// TIA Portal project "2022.04.27_指示灯依次亮灭" (V17)

(* hardware
DEVICE "S7-1500/ET200MP station_1"  S7-1500 station
   slot 0: "导轨_0"  Rack  6ES7 590-1***0-0AA0
   slot 1: "PLC_1"  CPU 1516-3 PN/DP  6ES7 516-3AN00-0AB0  V1.7
      slot 3: "CPU 显示_1"  6ES7591-1BA00-0AA0
      slot 32768: "PROFINET 接口_1"  X1
         slot 32769: "端口_1"  X1 P1
         slot 32770: "端口_2"  X1 P2
      slot 33024: "PROFINET 接口_2"  X2
         slot 33025: "端口_1"  X2 P1
      slot 33280: "DP 接口_1"  X3
   slot 2: "DI 32x24VDC BA_1"  DI 32x24VDC BA  6ES7 521-1BL10-0AA0  V1.1
   slot 3: "DQ 32x24VDC/0.5A HF_1"  DQ 32x24VDC/0.5A HF  6ES7 522-1BL01-0AB0  V1.1
*)

// ===== PLC "PLC_1"  CPU 1516-3 PN/DP =====

VAR_GLOBAL   // PLC tag table "默认变量表"
   "亮灯按钮" AT %I0.0 : Bool;
   "灭灯按钮" AT %I0.1 : Bool;
   "复位" AT %I0.2 : Bool;
   "按钮4" AT %I0.3 : Bool;
   "按钮5" AT %I0.4 : Bool;
   "按钮6" AT %I0.5 : Bool;
   "按钮7" AT %I0.6 : Bool;
   "按钮8" AT %I0.7 : Bool;
   "按钮9" AT %I1.0 : Bool;
   "按钮10" AT %I1.1 : Bool;
   "按钮11" AT %I1.2 : Bool;
   "指示灯1" AT %Q0.0 : Bool;
   "指示灯2" AT %Q0.1 : Bool;
   "指示灯3" AT %Q0.2 : Bool;
   "指示灯4" AT %Q0.3 : Bool;
   "指示灯5" AT %Q0.4 : Bool;
   "指示灯6" AT %Q0.5 : Bool;
   "指示灯7" AT %Q0.6 : Bool;
   "指示灯8" AT %Q0.7 : Bool;
   "指示灯9" AT %Q1.0 : Bool;
   "指示灯10" AT %Q1.1 : Bool;
   "指示灯11" AT %Q1.2 : Bool;
   "指示灯12" AT %Q1.3 : Bool;
END_VAR

DATA_BLOCK "计数亮灯LAD_DB"   // DB1
{ S7_Optimized_Access := 'TRUE' }
VERSION : 0.1
// stored: InstanceOfName 计数亮灯LAD
"计数亮灯LAD"
BEGIN
END_DATA_BLOCK

DATA_BLOCK "计数亮灯LAD_DB_1"   // DB3
{ S7_Optimized_Access := 'TRUE' }
VERSION : 0.1
// stored: InstanceOfName 计数亮灯LAD
"计数亮灯LAD"
BEGIN
END_DATA_BLOCK

DATA_BLOCK "计数亮灯FBD_DB"   // DB4
{ S7_Optimized_Access := 'TRUE' }
VERSION : 0.1
// stored: InstanceOfName 计数亮灯FBD
"计数亮灯FBD"
BEGIN
END_DATA_BLOCK

DATA_BLOCK "计数器SCL_DB"   // DB5
{ S7_Optimized_Access := 'TRUE' }
VERSION : 0.1
// stored: InstanceOfName 计数器SCL
"计数器SCL"
BEGIN
END_DATA_BLOCK

// folder: System blocks/Program resources

DATA_BLOCK "IEC_Counter_0_DB"   // DB2
{ S7_Optimized_Access := 'TRUE' }
AUTHOR : Simatic
FAMILY : IEC
NAME : CNTR
VERSION : 1.0
// stored: InstanceOfName IEC_COUNTER
"IEC_COUNTER"
BEGIN
END_DATA_BLOCK

// folder: (top level)

FUNCTION_BLOCK "计数亮灯LAD"   // FB1, LAD
{ S7_Optimized_Access := 'TRUE' }
VERSION : 0.1
   VAR RETAIN
      IEC_Counter_0_Instance : CTUD_INT;
      IEC_Counter_0_Instance_1 : CTUD_INT;
      IEC_Counter_0_Instance_2 : CTUD_INT;
      IEC_Counter_0_Instance_3 : CTUD_INT;
      IEC_Counter_0_Instance_4 : CTUD_INT;
      IEC_Counter_0_Instance_5 : CTUD_INT;
      IEC_Counter_0_Instance_6 : CTUD_INT;
      IEC_Counter_0_Instance_7 : CTUD_INT;
      IEC_Counter_0_Instance_8 : CTUD_INT;
      IEC_Counter_0_Instance_9 : CTUD_INT;
      IEC_Counter_0_Instance_10 : CTUD_INT;
      IEC_Counter_0_Instance_11 : CTD_INT;
   END_VAR
BEGIN

REGION Network 1: 亮灯按钮:选择置位，前灯亮和后灯不亮. 灭灯按钮：复位后灯依次不亮
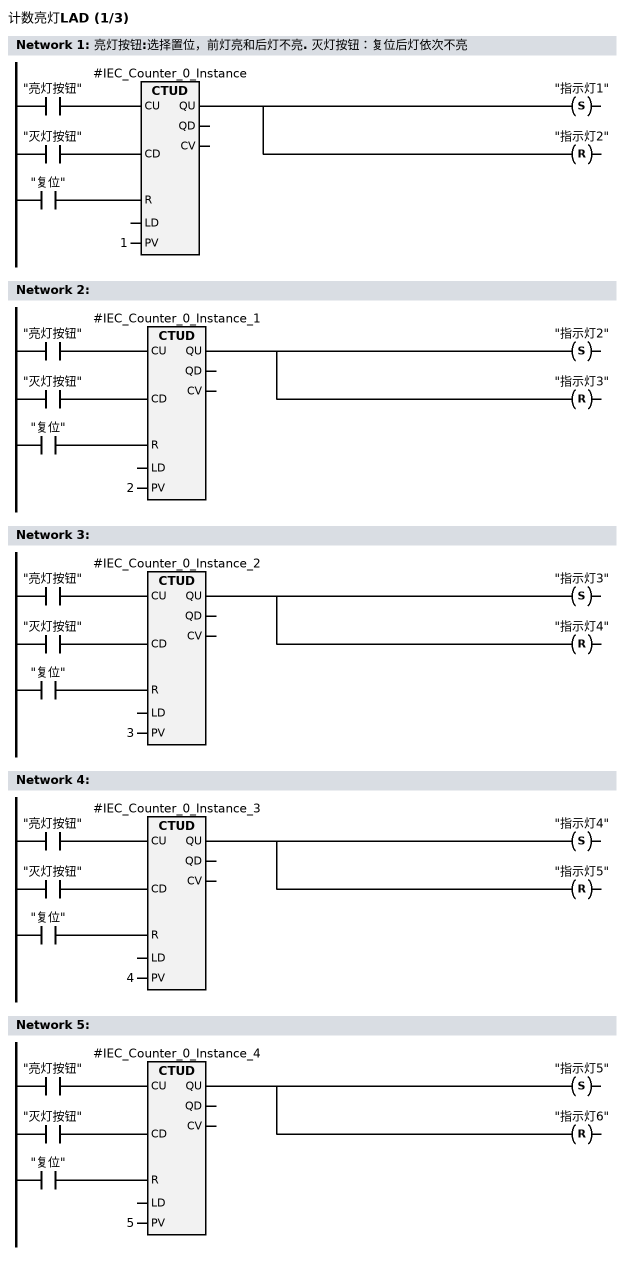
   #IEC_Counter_0_Instance(CU := "亮灯按钮", CD := "灭灯按钮", R := "复位", PV := 1);   // CTUD
   IF #IEC_Counter_0_Instance.QU THEN
       "指示灯1" := TRUE;
       "指示灯2" := FALSE;
   END_IF;
END_REGION

REGION Network 2
   #IEC_Counter_0_Instance_1(CU := "亮灯按钮", CD := "灭灯按钮", R := "复位", PV := 2);   // CTUD
   IF #IEC_Counter_0_Instance_1.QU THEN
       "指示灯2" := TRUE;
       "指示灯3" := FALSE;
   END_IF;
END_REGION

REGION Network 3
   #IEC_Counter_0_Instance_2(CU := "亮灯按钮", CD := "灭灯按钮", R := "复位", PV := 3);   // CTUD
   IF #IEC_Counter_0_Instance_2.QU THEN
       "指示灯3" := TRUE;
       "指示灯4" := FALSE;
   END_IF;
END_REGION

REGION Network 4
   #IEC_Counter_0_Instance_3(CU := "亮灯按钮", CD := "灭灯按钮", R := "复位", PV := 4);   // CTUD
   IF #IEC_Counter_0_Instance_3.QU THEN
       "指示灯4" := TRUE;
       "指示灯5" := FALSE;
   END_IF;
END_REGION

REGION Network 5
   #IEC_Counter_0_Instance_4(CU := "亮灯按钮", CD := "灭灯按钮", R := "复位", PV := 5);   // CTUD
   IF #IEC_Counter_0_Instance_4.QU THEN
       "指示灯5" := TRUE;
       "指示灯6" := FALSE;
   END_IF;
END_REGION

REGION Network 6
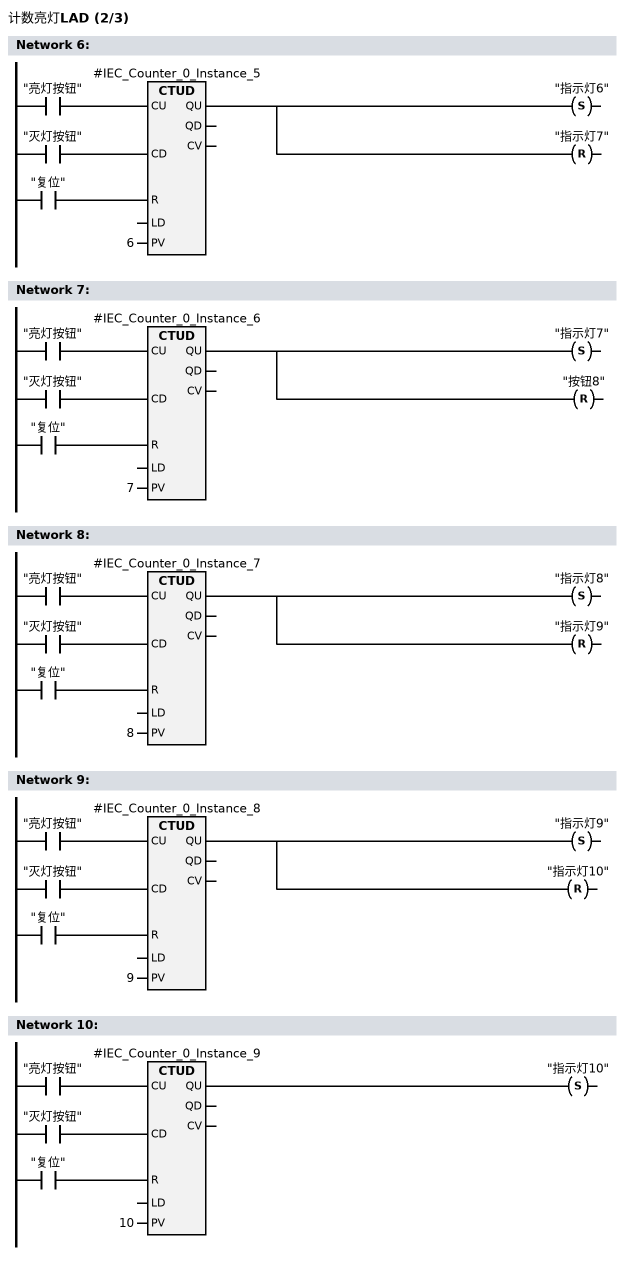
   #IEC_Counter_0_Instance_5(CU := "亮灯按钮", CD := "灭灯按钮", R := "复位", PV := 6);   // CTUD
   IF #IEC_Counter_0_Instance_5.QU THEN
       "指示灯6" := TRUE;
       "指示灯7" := FALSE;
   END_IF;
END_REGION

REGION Network 7
   #IEC_Counter_0_Instance_6(CU := "亮灯按钮", CD := "灭灯按钮", R := "复位", PV := 7);   // CTUD
   IF #IEC_Counter_0_Instance_6.QU THEN
       "指示灯7" := TRUE;
       "按钮8" := FALSE;
   END_IF;
END_REGION

REGION Network 8
   #IEC_Counter_0_Instance_7(CU := "亮灯按钮", CD := "灭灯按钮", R := "复位", PV := 8);   // CTUD
   IF #IEC_Counter_0_Instance_7.QU THEN
       "指示灯8" := TRUE;
       "指示灯9" := FALSE;
   END_IF;
END_REGION

REGION Network 9
   #IEC_Counter_0_Instance_8(CU := "亮灯按钮", CD := "灭灯按钮", R := "复位", PV := 9);   // CTUD
   IF #IEC_Counter_0_Instance_8.QU THEN
       "指示灯9" := TRUE;
       "指示灯10" := FALSE;
   END_IF;
END_REGION

REGION Network 10
   #IEC_Counter_0_Instance_9(CU := "亮灯按钮", CD := "灭灯按钮", R := "复位", PV := 10);   // CTUD
   IF #IEC_Counter_0_Instance_9.QU THEN "指示灯10" := TRUE; END_IF;
END_REGION

REGION Network 11: 复位指示灯1
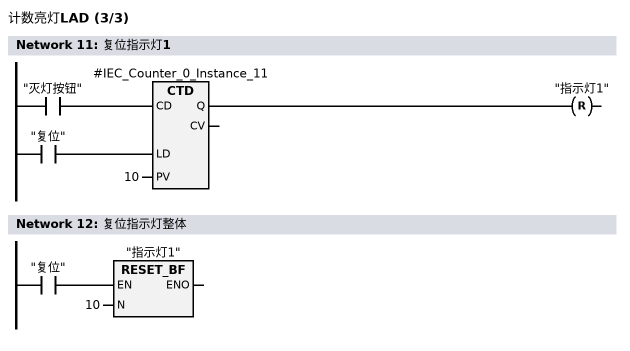
   #IEC_Counter_0_Instance_11(CD := "灭灯按钮", LD := "复位", PV := 10);   // CTD
   IF #IEC_Counter_0_Instance_11.Q THEN "指示灯1" := FALSE; END_IF;
END_REGION

REGION Network 12: 复位指示灯整体
   // no SCL statement known for RBitfield: written as a call
   IF "复位" THEN RESET_BF(operand := "指示灯1", n := 10); END_IF;
END_REGION
END_FUNCTION_BLOCK

FUNCTION_BLOCK "计数亮灯FBD"   // FB2, FBD
{ S7_Optimized_Access := 'TRUE' }
VERSION : 0.1
   VAR RETAIN
      IEC_Counter_0_Instance : CTUD_INT;
      IEC_Counter_0_Instance_1 : CTUD_INT;
      IEC_Counter_0_Instance_2 : CTUD_INT;
      IEC_Counter_0_Instance_3 : CTUD_INT;
      IEC_Counter_0_Instance_4 : CTUD_INT;
      IEC_Counter_0_Instance_5 : CTUD_INT;
      IEC_Counter_0_Instance_6 : CTUD_INT;
      IEC_Counter_0_Instance_7 : CTUD_INT;
      IEC_Counter_0_Instance_8 : CTUD_INT;
      IEC_Counter_0_Instance_9 : CTUD_INT;
      IEC_Counter_0_Instance_10 : CTD_INT;
   END_VAR
BEGIN

REGION Network 1
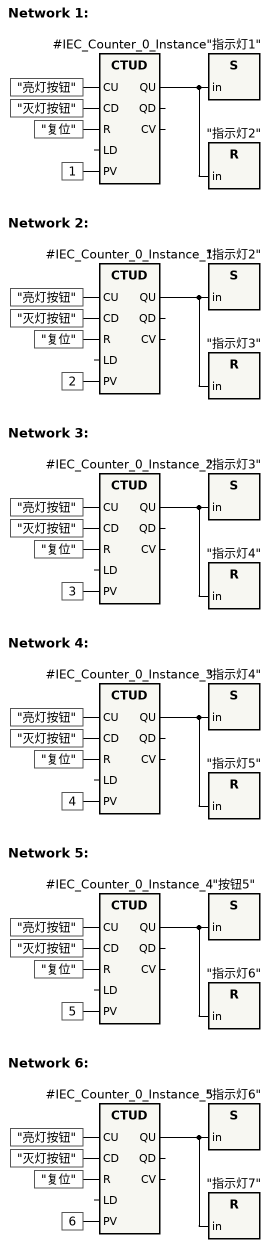
   #IEC_Counter_0_Instance(CU := "亮灯按钮", CD := "灭灯按钮", R := "复位", PV := 1);   // CTUD
   IF #IEC_Counter_0_Instance.QU THEN
       "指示灯1" := TRUE;
       "指示灯2" := FALSE;
   END_IF;
END_REGION

REGION Network 2
   #IEC_Counter_0_Instance_1(CU := "亮灯按钮", CD := "灭灯按钮", R := "复位", PV := 2);   // CTUD
   IF #IEC_Counter_0_Instance_1.QU THEN
       "指示灯2" := TRUE;
       "指示灯3" := FALSE;
   END_IF;
END_REGION

REGION Network 3
   #IEC_Counter_0_Instance_2(CU := "亮灯按钮", CD := "灭灯按钮", R := "复位", PV := 3);   // CTUD
   IF #IEC_Counter_0_Instance_2.QU THEN
       "指示灯3" := TRUE;
       "指示灯4" := FALSE;
   END_IF;
END_REGION

REGION Network 4
   #IEC_Counter_0_Instance_3(CU := "亮灯按钮", CD := "灭灯按钮", R := "复位", PV := 4);   // CTUD
   IF #IEC_Counter_0_Instance_3.QU THEN
       "指示灯4" := TRUE;
       "指示灯5" := FALSE;
   END_IF;
END_REGION

REGION Network 5
   #IEC_Counter_0_Instance_4(CU := "亮灯按钮", CD := "灭灯按钮", R := "复位", PV := 5);   // CTUD
   IF #IEC_Counter_0_Instance_4.QU THEN
       "按钮5" := TRUE;
       "指示灯6" := FALSE;
   END_IF;
END_REGION

REGION Network 6
   #IEC_Counter_0_Instance_5(CU := "亮灯按钮", CD := "灭灯按钮", R := "复位", PV := 6);   // CTUD
   IF #IEC_Counter_0_Instance_5.QU THEN
       "指示灯6" := TRUE;
       "指示灯7" := FALSE;
   END_IF;
END_REGION

REGION Network 7
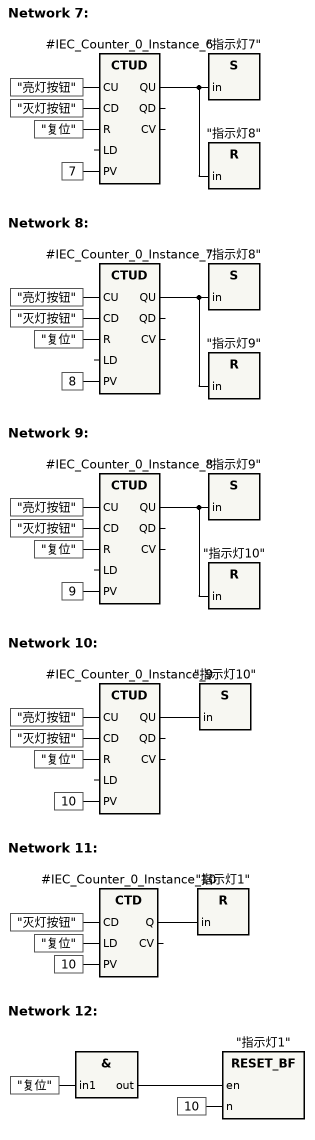
   #IEC_Counter_0_Instance_6(CU := "亮灯按钮", CD := "灭灯按钮", R := "复位", PV := 7);   // CTUD
   IF #IEC_Counter_0_Instance_6.QU THEN
       "指示灯7" := TRUE;
       "指示灯8" := FALSE;
   END_IF;
END_REGION

REGION Network 8
   #IEC_Counter_0_Instance_7(CU := "亮灯按钮", CD := "灭灯按钮", R := "复位", PV := 8);   // CTUD
   IF #IEC_Counter_0_Instance_7.QU THEN
       "指示灯8" := TRUE;
       "指示灯9" := FALSE;
   END_IF;
END_REGION

REGION Network 9
   #IEC_Counter_0_Instance_8(CU := "亮灯按钮", CD := "灭灯按钮", R := "复位", PV := 9);   // CTUD
   IF #IEC_Counter_0_Instance_8.QU THEN
       "指示灯9" := TRUE;
       "指示灯10" := FALSE;
   END_IF;
END_REGION

REGION Network 10
   #IEC_Counter_0_Instance_9(CU := "亮灯按钮", CD := "灭灯按钮", R := "复位", PV := 10);   // CTUD
   IF #IEC_Counter_0_Instance_9.QU THEN "指示灯10" := TRUE; END_IF;
END_REGION

REGION Network 11
   #IEC_Counter_0_Instance_10(CD := "灭灯按钮", LD := "复位", PV := 10);   // CTD
   IF #IEC_Counter_0_Instance_10.Q THEN "指示灯1" := FALSE; END_IF;
END_REGION

REGION Network 12
   // no SCL statement known for RBitfield: written as a call
   IF "复位" THEN RESET_BF(operand := "指示灯1", n := 10); END_IF;
END_REGION
END_FUNCTION_BLOCK

FUNCTION_BLOCK "计数器SCL"   // FB3, SCL
{ S7_Optimized_Access := 'TRUE' }
VERSION : 0.1
   VAR RETAIN
      IEC_Counter_0_Instance : CTUD_INT;
      IEC_Counter_0_Instance_1 : CTUD_INT;
      IEC_Counter_0_Instance_2 : CTUD_INT;
      IEC_Counter_0_Instance_3 : CTUD_INT;
      IEC_Counter_0_Instance_4 : CTUD_INT;
      IEC_Counter_0_Instance_5 : CTUD_INT;
      IEC_Counter_0_Instance_6 : CTUD_INT;
      IEC_Counter_0_Instance_7 : CTUD_INT;
      IEC_Counter_0_Instance_8 : CTUD_INT;
      IEC_Counter_0_Instance_9 : CTUD_INT;
      IEC_Counter_0_Instance_10 : CTD_INT;
   END_VAR
BEGIN
   //指示灯1复位
   #IEC_Counter_0_Instance_10(CD := "灭灯按钮",
                              LD := "复位",
                              PV := 10,
                              Q => "指示灯1");
   //复位指示灯程序
   IF "复位" THEN
       "指示灯1" := 0;
       "指示灯2" := 0;
       "指示灯3" := 0;
       "指示灯4" := 0;
       "指示灯5" := 0;
       "指示灯6" := 0;
       "指示灯7" := 0;
       "指示灯8" := 0;
       "指示灯9" := 0;
       "指示灯10" := 0;
   END_IF;

   //减法运算程序
   IF "指示灯1" THEN
       "指示灯2" := 0;
   END_IF;

   IF "指示灯2" THEN
       "指示灯3" := 0;
   END_IF;

   IF "指示灯3" THEN
       "指示灯4" := 0;
   END_IF;

   IF "指示灯4" THEN
       "指示灯5" := 0;
   END_IF;

   IF "指示灯5" THEN
       "指示灯6" := 0;
   END_IF;

   IF "指示灯6" THEN
       "指示灯7" := 0;
   END_IF;

   IF "指示灯7" THEN
       "指示灯8" := 0;
   END_IF;

   IF "指示灯8" THEN
       "指示灯9" := 0;
   END_IF;

   IF "指示灯9" THEN
       "指示灯10" := 0;
   END_IF;

   #IEC_Counter_0_Instance(CU:="亮灯按钮",
                           CD:="灭灯按钮",
                           R:="复位",
                           PV:=1,
                           QU=>"指示灯1");

   #IEC_Counter_0_Instance_1(CU:="亮灯按钮",
                             CD:="灭灯按钮",
                             R:="复位",
                             PV:=2,
                             QU=>"指示灯2");
   #IEC_Counter_0_Instance_2(CU:="亮灯按钮",
                             CD:="灭灯按钮",
                             R:="复位",
                             PV:=3,
                             QU=>"指示灯3");

   #IEC_Counter_0_Instance_3(CU := "亮灯按钮",
                             CD := "灭灯按钮",
                             R := "复位",
                             PV := 4,
                             QU => "指示灯4");

   #IEC_Counter_0_Instance_4(CU:="亮灯按钮",
                             CD:="灭灯按钮",
                             R:="复位",
                             PV:=5,
                             QU=>"指示灯5");

   #IEC_Counter_0_Instance_5(CU:="亮灯按钮",
                             CD:="灭灯按钮",
                             R:="复位",
                             PV:=6,
                             QU=>"指示灯6");

   #IEC_Counter_0_Instance_6(CU := "亮灯按钮",
                             CD := "灭灯按钮",
                             R := "复位",
                             PV := 7,
                             QU => "指示灯7");

   #IEC_Counter_0_Instance_7(CU := "亮灯按钮",
                             CD := "灭灯按钮",
                             R := "复位",
                             PV := 8,
                             QU => "指示灯8");

   #IEC_Counter_0_Instance_8(CU := "亮灯按钮",
                             CD := "灭灯按钮",
                             R := "复位",
                             PV := 9,
                             QU => "指示灯9");

   #IEC_Counter_0_Instance_9(CU := "亮灯按钮",
                             CD := "灭灯按钮",
                             R := "复位",
                             PV := 10,
                             QU => "指示灯10");
END_FUNCTION_BLOCK

ORGANIZATION_BLOCK "Main"   // OB1, LAD, ProgramCycle
TITLE = "Main Program Sweep (Cycle)"
{ S7_Optimized_Access := 'TRUE' }
VERSION : 0.1
   VAR_INPUT
      Initial_Call : Bool;   // Initial call of this OB
      Remanence : Bool;   // =True, if remanent data are available
   END_VAR
BEGIN

REGION Network 1
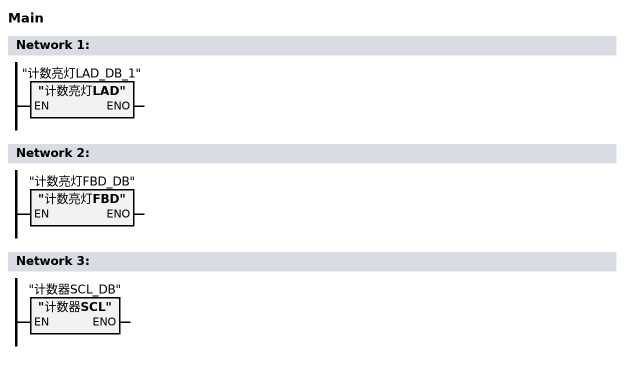
   RUNG wire#powerrail
      "计数亮灯LAD_DB_1"()
   END_RUNG
   // the same network as SCL:
   "计数亮灯LAD_DB_1"();   // "计数亮灯LAD"
END_REGION

REGION Network 2
   RUNG wire#powerrail
      "计数亮灯FBD_DB"()
   END_RUNG
   // the same network as SCL:
   "计数亮灯FBD_DB"();   // "计数亮灯FBD"
END_REGION

REGION Network 3
   RUNG wire#powerrail
      "计数器SCL_DB"()
   END_RUNG
   // the same network as SCL:
   "计数器SCL_DB"();   // "计数器SCL"
END_REGION
END_ORGANIZATION_BLOCK